KUKA KRL program: ps_602c3_bolha.src, ps_602c3_bolha.dat

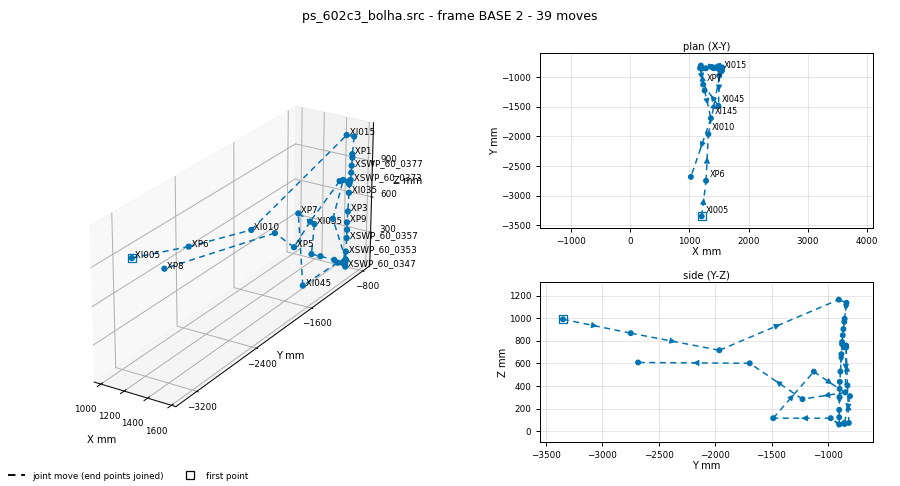
[picture p0: tool path of ps_602c3_bolha.src in frame BASE 2, 39 of 39 moves have a stored position in this frame; points joined in program order, loops and branches not executed]
--- ps_602c3_bolha.src ---
&ACCESS RVO1
&REL 1
&COMMENT Solda respot
&PARAM DISKPATH = KRC:\R1\Program
DEF ps_602c3_bolha( )

;FOLD INI
;FOLD SPOTTECH INI
USERSPOT(#INIT)
;ENDFOLD (SPOTTECH INI)
;FOLD GRIPPERTECH INI
USER_GRP(0,DUMMY,DUMMY,GDEFAULT)
;ENDFOLD (GRIPPERTECH INI)
  ;FOLD USER INI
    ;Make your modifications here

  ;ENDFOLD (USER INI)

   ;FOLD USER INI
      ;Make your modifications here
         ;FOLD COLLISION_V_3.01 INI
            IF (COLLISION_DATA[1].I_NR>0) THEN
               GLOBAL INTERRUPT DECL 21 WHEN $IN[COLLISION_DATA[1].I_NR]==FALSE DO COLLSTOP (1,0 )
            ENDIF
            IF (COLLISION_DATA[2].I_NR>0) THEN
               GLOBAL INTERRUPT DECL 22 WHEN $IN[COLLISION_DATA[2].I_NR]==FALSE DO COLLSTOP (2,0 )
            ENDIF
            IF (COLLISION_DATA[3].I_NR>0) THEN
               GLOBAL INTERRUPT DECL 23 WHEN $IN[COLLISION_DATA[3].I_NR]==FALSE DO COLLSTOP (3,0 )
            ENDIF
            IF (COLLISION_DATA[4].I_NR>0) THEN
               GLOBAL INTERRUPT DECL 24 WHEN $IN[COLLISION_DATA[4].I_NR]==FALSE DO COLLSTOP (4,0 )
            ENDIF
         ;ENDFOLD (COLLISION_V_3.01 INI)

   ;ENDFOLD (USER INI)
;ENDFOLD (INI)

; Caracterização dos meios de produção:
; Versão Atual:
; 15/05/2015 12:00 Name: P13.060-R1 CHANGES: Solda Geometrica Actros
; Gripper (INI;%{E}%V3.2.0,%MKUKATPGRIPPER,%CINIT,%VINIT,%P)

chk_w4_wechs_ok ( )           ; CHECK FERRAMENTA: C3

IF (NOT(GHOST())) THEN
IF MaxStandMenge (4) THEN
  MaxStandmengeErreicht (4)
ENDIF

IF Elektrodenwechsel (4) THEN
e_fraes_4()
ENDIF
ENDIF

;FOLD PTP l005  Vel=100 % P_OLP2 Tool[4]:Gun C03 Base[2]:Accelo;%{PE}%R8.2.20,%MKUKATPBASIS,%CMOVE,%VPTP,%P 1:PTP, 2:l005, 3:, 5:100, 7:P_OLP2
$BWDSTART = FALSE
PDAT_ACT= PP_OLP2
FDAT_ACT= Fl005
BAS(#PTP_PARAMS,100)
PTP Xl005
;ENDFOLD
;FOLD PTP P6 CONT Vel=100 % PDAT46 Tool[4]:PINCA C3 Base[2]:Accelo;%{PE}%R 8.2.20,%MKUKATPBASIS,%CMOVE,%VPTP,%P 1:PTP, 2:P6, 3:C_DIS, 5:100, 7:PDAT46
$BWDSTART=FALSE
PDAT_ACT=PPDAT46
FDAT_ACT=FP6
BAS(#PTP_PARAMS,100)
PTP XP6 C_DIS
;ENDFOLD
;FOLD PTP l010 Vel=100 % P_OLP3 Tool[4]:PINCA C3 Base[2]:Accelo;%{PE}%R 8.2.20,%MKUKATPBASIS,%CMOVE,%VPTP,%P 1:PTP, 2:l010, 3:, 5:100, 7:P_OLP3
$BWDSTART=FALSE
PDAT_ACT=PP_OLP3
FDAT_ACT=Fl010
BAS(#PTP_PARAMS,100)
PTP Xl010
;ENDFOLD

;FOLD OUT 3365 'R1_Solicita Lib. Soldar Geo1' State=TRUE ;%{PE}%R 8.2.20,%MKUKATPBASIS,%COUT,%VOUTX,%P 2:3365, 3:R1_Solicita Lib. Soldar Geo1, 5:TRUE, 6:
$OUT[3365]=TRUE
;ENDFOLD
;FOLD WAIT FOR ( IN 3323 'R1_Aguarda Lib. Soldar Respot GEO1' );%{PE}%R 8.2.20,%MKUKATPBASIS,%CEXT_WAIT_FOR,%VEXT_WAIT_FOR,%P 2:, 4:, 5:$IN, 6:3323, 7:R1_Aguarda Lib. Soldar Respot GEO1, 9:
WAIT FOR  ( $IN[3323] )
;ENDFOLD
;FOLD OUT 3331 'R1_Soldando' State=TRUE ;%{PE}%R 8.2.20,%MKUKATPBASIS,%COUT,%VOUTX,%P 2:3331, 3:R1_Soldando, 5:TRUE, 6:
$OUT[3331]=TRUE
;ENDFOLD
;FOLD OUT 3365 'R1_Solicita Lib. Soldar Geo1' State=FALSE ;%{PE}%R 8.2.20,%MKUKATPBASIS,%COUT,%VOUTX,%P 2:3365, 3:R1_Solicita Lib. Soldar Geo1, 5:FALSE, 6:
$OUT[3365]=FALSE
;ENDFOLD
;FOLD OUT 3369 'Area de Solda' State=FALSE ;%{PE}%R 8.2.20,%MKUKATPBASIS,%COUT,%VOUTX,%P 2:3369, 3:Area de Solda, 5:FALSE, 6:
$OUT[3369]=FALSE
;ENDFOLD

;FOLD PTP l015 CONT Vel=100 % PDAT1 Tool[4]:PINCA C3 Base[2]:Accelo;%{PE}%R 8.2.20,%MKUKATPBASIS,%CMOVE,%VPTP,%P 1:PTP, 2:l015, 3:C_DIS, 5:100, 7:PDAT1
$BWDSTART=FALSE
PDAT_ACT=PPDAT1
FDAT_ACT=Fl015
BAS(#PTP_PARAMS,100)
PTP Xl015 C_DIS
;ENDFOLD

;FOLD ; SWP_60_0385;%{PE}%R8.2.2,%MKUKATPSPOT,%CCOMMENT,%VNORMAL,%P 2:SWP_60_0385
;ENDFOLD
;FOLD PTP SWP_60_0385 PDAT2 SPOT Gun=3 RETR CLS PgNo1=151 ACTIVE=1 Tool[4]:PINCA C3 Base[2]:Accelo;%{PE}%R 8.2.2,%MKUKATPSPOT,%CSPOT,%VPTP,%P 1:PTP, 2:SWP_60_0385, 3:, 5:100, 7:PDAT2, 10:3, 12:#FIRST, 14:#CLO, 16:151, 18:1, 20:1, 22:0, 24:1, 25:NORMAL
$BWDSTART=FALSE
PDAT_ACT=PPDAT2
FDAT_ACT=FSWP_60_0385
BAS(#PTP_PARAMS,PPDAT2.VEL)
S_ACT.GUN=3
S_ACT.PAIR=SDEFAULT.PAIR
S_ACT.RETR=#CLO
S_ACT.CLO_TM=1
S_ACT.PGNO1=151
S_ACT.PGNO2=SDEFAULT.PGNO2
S_ACT.PRESS1=SDEFAULT.PRESS1
S_ACT.PRESS2=SDEFAULT.PRESS2
S_READY=FALSE
PTP XSWP_60_0385
USERSPOT(#SPOT, S_ACT)
WAIT FOR S_READY
;ENDFOLD

;FOLD PTP P1 CONT Vel=100 % PDAT7 Tool[4]:PINCA C3 Base[2]:Accelo;%{PE}%R 8.2.20,%MKUKATPBASIS,%CMOVE,%VPTP,%P 1:PTP, 2:P1, 3:C_DIS, 5:100, 7:PDAT7
$BWDSTART=FALSE
PDAT_ACT=PPDAT7
FDAT_ACT=FP1
BAS(#PTP_PARAMS,100)
PTP XP1 C_DIS
;ENDFOLD

;FOLD ; SWP_60_0379_1;%{PE}%R8.2.2,%MKUKATPSPOT,%CCOMMENT,%VNORMAL,%P 2:SWP_60_0379_1
;ENDFOLD
;FOLD PTP SWP_60_0379_1 PDAT6 SPOT Gun=3 RETR CLS PgNo1=153 ACTIVE=1 Tool[4]:PINCA C3 Base[2]:Accelo;%{PE}%R 8.2.2,%MKUKATPSPOT,%CSPOT,%VPTP,%P 1:PTP, 2:SWP_60_0379_1, 3:, 5:100, 7:PDAT6, 10:3, 12:#FIRST, 14:#CLO, 16:153, 18:1, 20:1, 22:0, 24:1, 25:NORMAL
$BWDSTART=FALSE
PDAT_ACT=PPDAT6
FDAT_ACT=FSWP_60_0379_1
BAS(#PTP_PARAMS,PPDAT6.VEL)
S_ACT.GUN=3
S_ACT.PAIR=SDEFAULT.PAIR
S_ACT.RETR=#CLO
S_ACT.CLO_TM=1
S_ACT.PGNO1=153
S_ACT.PGNO2=SDEFAULT.PGNO2
S_ACT.PRESS1=SDEFAULT.PRESS1
S_ACT.PRESS2=SDEFAULT.PRESS2
S_READY=FALSE
PTP XSWP_60_0379_1
USERSPOT(#SPOT, S_ACT)
WAIT FOR S_READY
;ENDFOLD

;FOLD ; SWP_60_0377;%{PE}%R8.2.2,%MKUKATPSPOT,%CCOMMENT,%VNORMAL,%P 2:SWP_60_0377
;ENDFOLD
;FOLD PTP SWP_60_0377 PDAT8 SPOT Gun=3 RETR CLS PgNo1=154 ACTIVE=1 Tool[4]:PINCA C3 Base[2]:Accelo;%{PE}%R 8.2.2,%MKUKATPSPOT,%CSPOT,%VPTP,%P 1:PTP, 2:SWP_60_0377, 3:, 5:100, 7:PDAT8, 10:3, 12:#FIRST, 14:#CLO, 16:154, 18:1, 20:1, 22:0, 24:1, 25:NORMAL
$BWDSTART=FALSE
PDAT_ACT=PPDAT8
FDAT_ACT=FSWP_60_0377
BAS(#PTP_PARAMS,PPDAT8.VEL)
S_ACT.GUN=3
S_ACT.PAIR=SDEFAULT.PAIR
S_ACT.RETR=#CLO
S_ACT.CLO_TM=1
S_ACT.PGNO1=154
S_ACT.PGNO2=SDEFAULT.PGNO2
S_ACT.PRESS1=SDEFAULT.PRESS1
S_ACT.PRESS2=SDEFAULT.PRESS2
S_READY=FALSE
PTP XSWP_60_0377
USERSPOT(#SPOT, S_ACT)
WAIT FOR S_READY
;ENDFOLD

;FOLD ; SWP_60_0375;%{PE}%R8.2.2,%MKUKATPSPOT,%CCOMMENT,%VNORMAL,%P 2:SWP_60_0375
;ENDFOLD
;FOLD PTP SWP_60_0375 PDAT9 SPOT Gun=3 RETR CLS PgNo1=155 ACTIVE=1 Tool[4]:PINCA C3 Base[2]:Accelo;%{PE}%R 8.2.2,%MKUKATPSPOT,%CSPOT,%VPTP,%P 1:PTP, 2:SWP_60_0375, 3:, 5:100, 7:PDAT9, 10:3, 12:#FIRST, 14:#CLO, 16:155, 18:1, 20:1, 22:0, 24:1, 25:NORMAL
$BWDSTART=FALSE
PDAT_ACT=PPDAT9
FDAT_ACT=FSWP_60_0375
BAS(#PTP_PARAMS,PPDAT9.VEL)
S_ACT.GUN=3
S_ACT.PAIR=SDEFAULT.PAIR
S_ACT.RETR=#CLO
S_ACT.CLO_TM=1
S_ACT.PGNO1=155
S_ACT.PGNO2=SDEFAULT.PGNO2
S_ACT.PRESS1=SDEFAULT.PRESS1
S_ACT.PRESS2=SDEFAULT.PRESS2
S_READY=FALSE
PTP XSWP_60_0375
USERSPOT(#SPOT, S_ACT)
WAIT FOR S_READY
;ENDFOLD

;FOLD ; SWP_60_0373;%{PE}%R8.2.2,%MKUKATPSPOT,%CCOMMENT,%VNORMAL,%P 2:SWP_60_0373
;ENDFOLD
;FOLD PTP SWP_60_0373 PDAT10 SPOT Gun=3 RETR CLS PgNo1=156 ACTIVE=1 Tool[4]:PINCA C3 Base[2]:Accelo;%{PE}%R 8.2.2,%MKUKATPSPOT,%CSPOT,%VPTP,%P 1:PTP, 2:SWP_60_0373, 3:, 5:100, 7:PDAT10, 10:3, 12:#FIRST, 14:#CLO, 16:156, 18:1, 20:1, 22:0, 24:1, 25:NORMAL
$BWDSTART=FALSE
PDAT_ACT=PPDAT10
FDAT_ACT=FSWP_60_0373
BAS(#PTP_PARAMS,PPDAT10.VEL)
S_ACT.GUN=3
S_ACT.PAIR=SDEFAULT.PAIR
S_ACT.RETR=#CLO
S_ACT.CLO_TM=1
S_ACT.PGNO1=156
S_ACT.PGNO2=SDEFAULT.PGNO2
S_ACT.PRESS1=SDEFAULT.PRESS1
S_ACT.PRESS2=SDEFAULT.PRESS2
S_READY=FALSE
PTP XSWP_60_0373
USERSPOT(#SPOT, S_ACT)
WAIT FOR S_READY
;ENDFOLD

;FOLD PTP P10 CONT Vel=100 % PDAT50 Tool[4]:PINCA C3 Base[2]:Accelo;%{PE}%R 8.2.20,%MKUKATPBASIS,%CMOVE,%VPTP,%P 1:PTP, 2:P10, 3:C_DIS, 5:100, 7:PDAT50
$BWDSTART=FALSE
PDAT_ACT=PPDAT50
FDAT_ACT=FP10
BAS(#PTP_PARAMS,100)
PTP XP10 C_DIS
;ENDFOLD
;FOLD PTP l035 CONT Vel=100 % PDAT11 Tool[4]:PINCA C3 Base[2]:Accelo;%{PE}%R 8.2.20,%MKUKATPBASIS,%CMOVE,%VPTP,%P 1:PTP, 2:l035, 3:C_DIS, 5:100, 7:PDAT11
$BWDSTART=FALSE
PDAT_ACT=PPDAT11
FDAT_ACT=Fl035
BAS(#PTP_PARAMS,100)
PTP Xl035 C_DIS
;ENDFOLD
;FOLD PTP P3 CONT Vel=100 % PDAT15 Tool[4]:PINCA C3 Base[2]:Accelo;%{PE}%R 8.2.20,%MKUKATPBASIS,%CMOVE,%VPTP,%P 1:PTP, 2:P3, 3:C_DIS, 5:100, 7:PDAT15
$BWDSTART=FALSE
PDAT_ACT=PPDAT15
FDAT_ACT=FP3
BAS(#PTP_PARAMS,100)
PTP XP3 C_DIS
;ENDFOLD
;FOLD PTP P9 CONT Vel=100 % PDAT49 Tool[4]:PINCA C3 Base[2]:Accelo;%{PE}%R 8.2.20,%MKUKATPBASIS,%CMOVE,%VPTP,%P 1:PTP, 2:P9, 3:C_DIS, 5:100, 7:PDAT49
$BWDSTART=FALSE
PDAT_ACT=PPDAT49
FDAT_ACT=FP9
BAS(#PTP_PARAMS,100)
PTP XP9 C_DIS
;ENDFOLD

;FOLD ; SWP_60_0359;%{PE}%R8.2.2,%MKUKATPSPOT,%CCOMMENT,%VNORMAL,%P 2:SWP_60_0359
;ENDFOLD
;FOLD PTP SWP_60_0359 PDAT16 SPOT Gun=3 RETR CLS PgNo1=158 ACTIVE=1 Tool[4]:PINCA C3 Base[2]:Accelo;%{PE}%R 8.2.2,%MKUKATPSPOT,%CSPOT,%VPTP,%P 1:PTP, 2:SWP_60_0359, 3:, 5:100, 7:PDAT16, 10:3, 12:#FIRST, 14:#CLO, 16:158, 18:1, 20:1, 22:0, 24:1, 25:NORMAL
$BWDSTART=FALSE
PDAT_ACT=PPDAT16
FDAT_ACT=FSWP_60_0359
BAS(#PTP_PARAMS,PPDAT16.VEL)
S_ACT.GUN=3
S_ACT.PAIR=SDEFAULT.PAIR
S_ACT.RETR=#CLO
S_ACT.CLO_TM=1
S_ACT.PGNO1=158
S_ACT.PGNO2=SDEFAULT.PGNO2
S_ACT.PRESS1=SDEFAULT.PRESS1
S_ACT.PRESS2=SDEFAULT.PRESS2
S_READY=FALSE
PTP XSWP_60_0359
USERSPOT(#SPOT, S_ACT)
WAIT FOR S_READY
;ENDFOLD

;FOLD ; SWP_60_0357;%{PE}%R8.2.2,%MKUKATPSPOT,%CCOMMENT,%VNORMAL,%P 2:SWP_60_0357
;ENDFOLD
;FOLD PTP SWP_60_0357 PDAT17 SPOT Gun=3 RETR CLS PgNo1=159 ACTIVE=1 Tool[4]:PINCA C3 Base[2]:Accelo;%{PE}%R 8.2.2,%MKUKATPSPOT,%CSPOT,%VPTP,%P 1:PTP, 2:SWP_60_0357, 3:, 5:100, 7:PDAT17, 10:3, 12:#FIRST, 14:#CLO, 16:159, 18:1, 20:1, 22:0, 24:1, 25:NORMAL
$BWDSTART=FALSE
PDAT_ACT=PPDAT17
FDAT_ACT=FSWP_60_0357
BAS(#PTP_PARAMS,PPDAT17.VEL)
S_ACT.GUN=3
S_ACT.PAIR=SDEFAULT.PAIR
S_ACT.RETR=#CLO
S_ACT.CLO_TM=1
S_ACT.PGNO1=159
S_ACT.PGNO2=SDEFAULT.PGNO2
S_ACT.PRESS1=SDEFAULT.PRESS1
S_ACT.PRESS2=SDEFAULT.PRESS2
S_READY=FALSE
PTP XSWP_60_0357
USERSPOT(#SPOT, S_ACT)
WAIT FOR S_READY
;ENDFOLD

;FOLD ; SWP_60_0353;%{PE}%R8.2.2,%MKUKATPSPOT,%CCOMMENT,%VNORMAL,%P 2:SWP_60_0353
;ENDFOLD
;FOLD PTP SWP_60_0353 PDAT18 SPOT Gun=3 RETR CLS PgNo1=160 ACTIVE=1 Tool[4]:PINCA C3 Base[2]:Accelo;%{PE}%R 8.2.2,%MKUKATPSPOT,%CSPOT,%VPTP,%P 1:PTP, 2:SWP_60_0353, 3:, 5:100, 7:PDAT18, 10:3, 12:#FIRST, 14:#CLO, 16:160, 18:1, 20:1, 22:0, 24:1, 25:NORMAL
$BWDSTART=FALSE
PDAT_ACT=PPDAT18
FDAT_ACT=FSWP_60_0353
BAS(#PTP_PARAMS,PPDAT18.VEL)
S_ACT.GUN=3
S_ACT.PAIR=SDEFAULT.PAIR
S_ACT.RETR=#CLO
S_ACT.CLO_TM=1
S_ACT.PGNO1=160
S_ACT.PGNO2=SDEFAULT.PGNO2
S_ACT.PRESS1=SDEFAULT.PRESS1
S_ACT.PRESS2=SDEFAULT.PRESS2
S_READY=FALSE
PTP XSWP_60_0353
USERSPOT(#SPOT, S_ACT)
WAIT FOR S_READY
;ENDFOLD

;FOLD ; SWP_60_0351;%{PE}%R8.2.2,%MKUKATPSPOT,%CCOMMENT,%VNORMAL,%P 2:SWP_60_0351
;ENDFOLD
;FOLD PTP SWP_60_0351 PDAT19 SPOT Gun=3 RETR CLS PgNo1=161 ACTIVE=1 Tool[4]:PINCA C3 Base[2]:Accelo;%{PE}%R 8.2.2,%MKUKATPSPOT,%CSPOT,%VPTP,%P 1:PTP, 2:SWP_60_0351, 3:, 5:100, 7:PDAT19, 10:3, 12:#FIRST, 14:#CLO, 16:161, 18:1, 20:1, 22:0, 24:1, 25:NORMAL
$BWDSTART=FALSE
PDAT_ACT=PPDAT19
FDAT_ACT=FSWP_60_0351
BAS(#PTP_PARAMS,PPDAT19.VEL)
S_ACT.GUN=3
S_ACT.PAIR=SDEFAULT.PAIR
S_ACT.RETR=#CLO
S_ACT.CLO_TM=1
S_ACT.PGNO1=161
S_ACT.PGNO2=SDEFAULT.PGNO2
S_ACT.PRESS1=SDEFAULT.PRESS1
S_ACT.PRESS2=SDEFAULT.PRESS2
S_READY=FALSE
PTP XSWP_60_0351
USERSPOT(#SPOT, S_ACT)
WAIT FOR S_READY
;ENDFOLD

;FOLD ; SWP_60_0347;%{PE}%R8.2.2,%MKUKATPSPOT,%CCOMMENT,%VNORMAL,%P 2:SWP_60_0347
;ENDFOLD
;FOLD PTP SWP_60_0347 PDAT20 SPOT Gun=3 RETR OPN PgNo1=162 ACTIVE=1 Tool[4]:PINCA C3 Base[2]:Accelo;%{PE}%R 8.2.2,%MKUKATPSPOT,%CSPOT,%VPTP,%P 1:PTP, 2:SWP_60_0347, 3:, 5:100, 7:PDAT20, 10:3, 12:#FIRST, 14:#OPN, 16:162, 18:1, 20:0, 22:0, 24:1, 25:NORMAL
$BWDSTART=FALSE
PDAT_ACT=PPDAT20
FDAT_ACT=FSWP_60_0347
BAS(#PTP_PARAMS,PPDAT20.VEL)
S_ACT.GUN=3
S_ACT.PAIR=SDEFAULT.PAIR
S_ACT.RETR=#OPN
S_ACT.CLO_TM=1
S_ACT.PGNO1=162
S_ACT.PGNO2=SDEFAULT.PGNO2
S_ACT.PRESS1=SDEFAULT.PRESS1
S_ACT.PRESS2=SDEFAULT.PRESS2
S_READY=FALSE
PTP XSWP_60_0347
USERSPOT(#SPOT, S_ACT)
WAIT FOR S_READY
;ENDFOLD

;FOLD PTP l040 CONT Vel=100 % PDAT21 Tool[4]:PINCA C3 Base[2]:Accelo;%{PE}%R 8.2.20,%MKUKATPBASIS,%CMOVE,%VPTP,%P 1:PTP, 2:l040, 3:C_DIS, 5:100, 7:PDAT21
$BWDSTART=FALSE
PDAT_ACT=PPDAT21
FDAT_ACT=Fl040
BAS(#PTP_PARAMS,100)
PTP Xl040 C_DIS
;ENDFOLD
;FOLD PTP l045 Vel=100 % PDAT22 Tool[4]:PINCA C3 Base[2]:Accelo;%{PE}%R 8.2.20,%MKUKATPBASIS,%CMOVE,%VPTP,%P 1:PTP, 2:l045, 3:, 5:100, 7:PDAT22
$BWDSTART=FALSE
PDAT_ACT=PPDAT22
FDAT_ACT=Fl045
BAS(#PTP_PARAMS,100)
PTP Xl045
;ENDFOLD

;FOLD Collision.Monitoring_3_On ;%{PE}%MKUKATPUSER
COLLSTOP( 3, 1 ) ;Interrupt-Controlled
;ENDFOLD

;FOLD PTP P7 CONT Vel=100 % PDAT47 Tool[4]:PINCA C3 Base[2]:Accelo;%{PE}%R 8.2.20,%MKUKATPBASIS,%CMOVE,%VPTP,%P 1:PTP, 2:P7, 3:C_DIS, 5:100, 7:PDAT47
$BWDSTART=FALSE
PDAT_ACT=PPDAT47
FDAT_ACT=FP7
BAS(#PTP_PARAMS,100)
PTP XP7 C_DIS
;ENDFOLD
;FOLD PTP l055 CONT Vel=100 % PDAT23 Tool[4]:PINCA C3 Base[2]:Accelo;%{PE}%R 8.2.20,%MKUKATPBASIS,%CMOVE,%VPTP,%P 1:PTP, 2:l055, 3:C_DIS, 5:100, 7:PDAT23
$BWDSTART=FALSE
PDAT_ACT=PPDAT23
FDAT_ACT=Fl055
BAS(#PTP_PARAMS,100)
PTP Xl055 C_DIS
;ENDFOLD

;FOLD ; SWP_60_0329;%{PE}%R8.2.2,%MKUKATPSPOT,%CCOMMENT,%VNORMAL,%P 2:SWP_60_0329
;ENDFOLD
;FOLD PTP SWP_60_0329 PDAT25 SPOT Gun=3 RETR CLS PgNo1=163 ACTIVE=1 Tool[4]:PINCA C3 Base[2]:Accelo;%{PE}%R 8.2.2,%MKUKATPSPOT,%CSPOT,%VPTP,%P 1:PTP, 2:SWP_60_0329, 3:, 5:100, 7:PDAT25, 10:3, 12:#FIRST, 14:#CLO, 16:163, 18:1, 20:0, 22:0, 24:1, 25:NORMAL
$BWDSTART=FALSE
PDAT_ACT=PPDAT25
FDAT_ACT=FSWP_60_0329
BAS(#PTP_PARAMS,PPDAT25.VEL)
S_ACT.GUN=3
S_ACT.PAIR=SDEFAULT.PAIR
S_ACT.RETR=#CLO
S_ACT.CLO_TM=1
S_ACT.PGNO1=163
S_ACT.PGNO2=SDEFAULT.PGNO2
S_ACT.PRESS1=SDEFAULT.PRESS1
S_ACT.PRESS2=SDEFAULT.PRESS2
S_READY=FALSE
PTP XSWP_60_0329
USERSPOT(#SPOT, S_ACT)
WAIT FOR S_READY
;ENDFOLD

;FOLD PTP l065 CONT Vel=100 % PDAT26 Tool[4]:PINCA C3 Base[2]:Accelo;%{PE}%R 8.2.20,%MKUKATPBASIS,%CMOVE,%VPTP,%P 1:PTP, 2:l065, 3:C_DIS, 5:100, 7:PDAT26
$BWDSTART=FALSE
PDAT_ACT=PPDAT26
FDAT_ACT=Fl065
BAS(#PTP_PARAMS,100)
PTP Xl065 C_DIS
;ENDFOLD
;FOLD PTP l070 CONT Vel=100 % PDAT27 Tool[4]:PINCA C3 Base[2]:Accelo;%{PE}%R 8.2.20,%MKUKATPBASIS,%CMOVE,%VPTP,%P 1:PTP, 2:l070, 3:C_DIS, 5:100, 7:PDAT27
$BWDSTART=FALSE
PDAT_ACT=PPDAT27
FDAT_ACT=Fl070
BAS(#PTP_PARAMS,100)
PTP Xl070 C_DIS
;ENDFOLD

;FOLD ; SWP_60_0343;%{PE}%R8.2.2,%MKUKATPSPOT,%CCOMMENT,%VNORMAL,%P 2:SWP_60_0343
;ENDFOLD
;FOLD PTP SWP_60_0343 PDAT28 SPOT Gun=3 RETR CLS PgNo1=165 ACTIVE=1 Tool[4]:PINCA C3 Base[2]:Accelo;%{PE}%R 8.2.2,%MKUKATPSPOT,%CSPOT,%VPTP,%P 1:PTP, 2:SWP_60_0343, 3:, 5:100, 7:PDAT28, 10:3, 12:#FIRST, 14:#CLO, 16:165, 18:1, 20:0, 22:0, 24:1, 25:NORMAL
$BWDSTART=FALSE
PDAT_ACT=PPDAT28
FDAT_ACT=FSWP_60_0343
BAS(#PTP_PARAMS,PPDAT28.VEL)
S_ACT.GUN=3
S_ACT.PAIR=SDEFAULT.PAIR
S_ACT.RETR=#CLO
S_ACT.CLO_TM=1
S_ACT.PGNO1=165
S_ACT.PGNO2=SDEFAULT.PGNO2
S_ACT.PRESS1=SDEFAULT.PRESS1
S_ACT.PRESS2=SDEFAULT.PRESS2
S_READY=FALSE
PTP XSWP_60_0343
USERSPOT(#SPOT, S_ACT)
WAIT FOR S_READY
;ENDFOLD

;FOLD ; SWP_60_0345;%{PE}%R8.2.2,%MKUKATPSPOT,%CCOMMENT,%VNORMAL,%P 2:SWP_60_0345
;ENDFOLD
;FOLD PTP SWP_60_0345 PDAT29 SPOT Gun=3 RETR OPN PgNo1=164 ACTIVE=1 Tool[4]:PINCA C3 Base[2]:Accelo;%{PE}%R 8.2.2,%MKUKATPSPOT,%CSPOT,%VPTP,%P 1:PTP, 2:SWP_60_0345, 3:, 5:100, 7:PDAT29, 10:3, 12:#FIRST, 14:#OPN, 16:164, 18:1, 20:0, 22:0, 24:1, 25:NORMAL
$BWDSTART=FALSE
PDAT_ACT=PPDAT29
FDAT_ACT=FSWP_60_0345
BAS(#PTP_PARAMS,PPDAT29.VEL)
S_ACT.GUN=3
S_ACT.PAIR=SDEFAULT.PAIR
S_ACT.RETR=#OPN
S_ACT.CLO_TM=1
S_ACT.PGNO1=164
S_ACT.PGNO2=SDEFAULT.PGNO2
S_ACT.PRESS1=SDEFAULT.PRESS1
S_ACT.PRESS2=SDEFAULT.PRESS2
S_READY=FALSE
PTP XSWP_60_0345
USERSPOT(#SPOT, S_ACT)
WAIT FOR S_READY
;ENDFOLD

;FOLD PTP l075 CONT Vel=100 % PDAT30 Tool[4]:PINCA C3 Base[2]:Accelo;%{PE}%R 8.2.20,%MKUKATPBASIS,%CMOVE,%VPTP,%P 1:PTP, 2:l075, 3:C_DIS, 5:100, 7:PDAT30
$BWDSTART=FALSE
PDAT_ACT=PPDAT30
FDAT_ACT=Fl075
BAS(#PTP_PARAMS,100)
PTP Xl075 C_DIS
;ENDFOLD
;FOLD PTP l080 CONT Vel=100 % PDAT31 Tool[4]:PINCA C3 Base[2]:Accelo;%{PE}%R 8.2.20,%MKUKATPBASIS,%CMOVE,%VPTP,%P 1:PTP, 2:l080, 3:C_DIS, 5:100, 7:PDAT31
$BWDSTART=FALSE
PDAT_ACT=PPDAT31
FDAT_ACT=Fl080
BAS(#PTP_PARAMS,100)
PTP Xl080 C_DIS
;ENDFOLD
;FOLD PTP l110 CONT Vel=100 % PDAT39 Tool[4]:PINCA C3 Base[2]:Accelo;%{PE}%R 8.2.20,%MKUKATPBASIS,%CMOVE,%VPTP,%P 1:PTP, 2:l110, 3:C_DIS, 5:100, 7:PDAT39
$BWDSTART=FALSE
PDAT_ACT=PPDAT39
FDAT_ACT=Fl110
BAS(#PTP_PARAMS,100)
PTP Xl110 C_DIS
;ENDFOLD
;FOLD PTP l115 CONT Vel=100 % PDAT40 Tool[4]:PINCA C3 Base[2]:Accelo;%{PE}%R 8.2.20,%MKUKATPBASIS,%CMOVE,%VPTP,%P 1:PTP, 2:l115, 3:C_DIS, 5:100, 7:PDAT40
$BWDSTART=FALSE
PDAT_ACT=PPDAT40
FDAT_ACT=Fl115
BAS(#PTP_PARAMS,100)
PTP Xl115 C_DIS
;ENDFOLD

;FOLD ; SWP_60_0401;%{PE}%R8.2.2,%MKUKATPSPOT,%CCOMMENT,%VNORMAL,%P 2:SWP_60_0401
;ENDFOLD
;FOLD PTP SWP_60_0401 PDAT41 SPOT Gun=3 RETR OPN PgNo1=168 ACTIVE=1 Tool[4]:PINCA C3 Base[2]:Accelo;%{PE}%R 8.2.2,%MKUKATPSPOT,%CSPOT,%VPTP,%P 1:PTP, 2:SWP_60_0401, 3:, 5:100, 7:PDAT41, 10:3, 12:#FIRST, 14:#OPN, 16:168, 18:1, 20:0, 22:0, 24:1, 25:NORMAL
$BWDSTART=FALSE
PDAT_ACT=PPDAT41
FDAT_ACT=FSWP_60_0401
BAS(#PTP_PARAMS,PPDAT41.VEL)
S_ACT.GUN=3
S_ACT.PAIR=SDEFAULT.PAIR
S_ACT.RETR=#OPN
S_ACT.CLO_TM=1
S_ACT.PGNO1=168
S_ACT.PGNO2=SDEFAULT.PGNO2
S_ACT.PRESS1=SDEFAULT.PRESS1
S_ACT.PRESS2=SDEFAULT.PRESS2
S_READY=FALSE
PTP XSWP_60_0401
USERSPOT(#SPOT, S_ACT)
WAIT FOR S_READY
;ENDFOLD

;FOLD PTP l120 CONT Vel=100 % PDAT42 Tool[4]:PINCA C3 Base[2]:Accelo;%{PE}%R 8.2.20,%MKUKATPBASIS,%CMOVE,%VPTP,%P 1:PTP, 2:l120, 3:C_DIS, 5:100, 7:PDAT42
$BWDSTART=FALSE
PDAT_ACT=PPDAT42
FDAT_ACT=Fl120
BAS(#PTP_PARAMS,100)
PTP Xl120 C_DIS
;ENDFOLD
;FOLD PTP l125 CONT Vel=100 % PDAT43 Tool[4]:PINCA C3 Base[2]:Accelo;%{PE}%R 8.2.20,%MKUKATPBASIS,%CMOVE,%VPTP,%P 1:PTP, 2:l125, 3:C_DIS, 5:100, 7:PDAT43
$BWDSTART=FALSE
PDAT_ACT=PPDAT43
FDAT_ACT=Fl125
BAS(#PTP_PARAMS,100)
PTP Xl125 C_DIS
;ENDFOLD
;FOLD PTP l135 CONT Vel=100 % P_OLP6 Tool[4]:PINCA C3 Base[2]:Accelo;%{PE}%R 8.2.20,%MKUKATPBASIS,%CMOVE,%VPTP,%P 1:PTP, 2:l135, 3:C_DIS, 5:100, 7:P_OLP6
$BWDSTART=FALSE
PDAT_ACT=PP_OLP6
FDAT_ACT=Fl135
BAS(#PTP_PARAMS,100)
PTP Xl135 C_DIS
;ENDFOLD
;FOLD PTP P5 CONT Vel=100 % PDAT45 Tool[4]:PINCA C3 Base[2]:Accelo;%{PE}%R 8.2.20,%MKUKATPBASIS,%CMOVE,%VPTP,%P 1:PTP, 2:P5, 3:C_DIS, 5:100, 7:PDAT45
$BWDSTART=FALSE
PDAT_ACT=PPDAT45
FDAT_ACT=FP5
BAS(#PTP_PARAMS,100)
PTP XP5 C_DIS
;ENDFOLD
;FOLD PTP l145 CONT Vel=100 % P_OLP8 Tool[4]:PINCA C3 Base[2]:Accelo;%{PE}%R 8.2.20,%MKUKATPBASIS,%CMOVE,%VPTP,%P 1:PTP, 2:l145, 3:C_DIS, 5:100, 7:P_OLP8
$BWDSTART=FALSE
PDAT_ACT=PP_OLP8
FDAT_ACT=Fl145
BAS(#PTP_PARAMS,100)
PTP Xl145 C_DIS
;ENDFOLD

;FOLD OUT 3331 'R1_Soldando' State=FALSE ;%{PE}%R 8.2.20,%MKUKATPBASIS,%COUT,%VOUTX,%P 2:3331, 3:R1_Soldando, 5:FALSE, 6:
$OUT[3331]=FALSE
;ENDFOLD
;FOLD OUT 3369 'Area de Solda' State=TRUE ;%{PE}%R 8.2.20,%MKUKATPBASIS,%COUT,%VOUTX,%P 2:3369, 3:Area de Solda, 5:TRUE, 6:
$OUT[3369]=TRUE
;ENDFOLD

;FOLD PULSE 3367 'R1_Solda Respot Geo1 OK' State=TRUE Time=3 sec;%{PE}%R 8.2.20,%MKUKATPBASIS,%COUT,%VPULSE,%P 2:3367, 3:R1_Solda Respot Geo1 OK, 5:TRUE, 6:, 8:3
PULSE($OUT[3367], TRUE,3)
;ENDFOLD

;FOLD PTP P8 Vel=100 % PDAT48 Tool[4]:PINCA C3 Base[2]:Accelo;%{PE}%R 8.2.20,%MKUKATPBASIS,%CMOVE,%VPTP,%P 1:PTP, 2:P8, 3:, 5:100, 7:PDAT48
$BWDSTART=FALSE
PDAT_ACT=PPDAT48
FDAT_ACT=FP8
BAS(#PTP_PARAMS,100)
PTP XP8
;ENDFOLD

IF (NOT(GHOST())) THEN
IF FraesAnf(4) THEN
f_fraes_4()
ENDIF
ENDIF

END

--- ps_602c3_bolha.dat ---
&ACCESS RVO1
&REL 1
&COMMENT Solda respot
&PARAM DISKPATH = KRC:\R1\Program
DEFDAT  ps_602c3_bolha
;FOLD EXTERNAL DECLARATIONS;%{PE}%MKUKATPBASIS,%CEXT,%VCOMMON,%P
;FOLD GRIPPERTECH EXT
EXT  H50 (INT  :IN,INT  :IN,INT  :IN,GRP_TYP  :IN )
;ENDFOLD (GRIPPERTECH EXT)
;FOLD SPOTTECH EXT
EXT  USERSPOT (S_COMMAND  :IN,SPOT_TYPE  :IN )
;ENDFOLD (SPOTTECH EXT)
;FOLD BASISTECH EXT;%{PE}%MKUKATPBASIS,%CEXT,%VEXT,%P
EXT  BAS (BAS_COMMAND  :IN,REAL  :IN )
DECL INT SUCCESS
;ENDFOLD (BASISTECH EXT)
;FOLD USER EXT;%{E}%MKUKATPUSER,%CEXT,%VEXT,%P
;Make your modifications here

;ENDFOLD (USER EXT)
;ENDFOLD (EXTERNAL DECLARATIONS)
DECL FDAT FLO1077={TOOL_NO 4,BASE_NO 2,IPO_FRAME #BASE,POINT2[] " "}
DECL PDAT PP_OLP1={VEL 100.0,ACC 50.0,APO_DIST 0.0}
DECL FDAT Fl005={TOOL_NO 4,BASE_NO 2,IPO_FRAME #BASE,POINT2[] " "}
DECL PDAT PP_OLP2={VEL 100.0,ACC 50.0,APO_DIST 0.0}
DECL E6POS Xl005={X 1207.93994,Y -3347.26807,Z 991.342712,A 123.692596,B -61.2644691,C 128.996994,S 18,T 3,E1 0.0,E2 0.0,E3 0.0,E4 0.0,E5 0.0,E6 0.0}
DECL FDAT Fl010={TOOL_NO 4,BASE_NO 2,IPO_FRAME #BASE,POINT2[] " "}
DECL PDAT PP_OLP3={VEL 100.0,ACC 100.0,APO_DIST 10.0,APO_MODE #CDIS}
DECL E6POS Xl010={X 1321.125,Y -1961.92896,Z 716.955383,A 162.414505,B -50.7519913,C 56.327549,S 18,T 3,E1 0.0,E2 0.0,E3 0.0,E4 0.0,E5 0.0,E6 0.0}
DECL FDAT Fl015={TOOL_NO 4,BASE_NO 2,IPO_FRAME #BASE,POINT2[] " "}
DECL E6POS Xl015={X 1525.30005,Y -903.920776,Z 1165.68701,A 79.9386902,B -67.3189468,C 102.332298,S 18,T 3,E1 0.0,E2 0.0,E3 0.0,E4 0.0,E5 0.0,E6 0.0}
DECL LDAT LL_OLP1={VEL 2.0,ACC 23.0,APO_DIST 0.0,APO_FAC 0.0,ORI_TYP #VAR,CIRC_TYP #BASE,JERK_FAC 50.0}
DECL FDAT FSWP_60_0387={TOOL_NO 4,BASE_NO 2,IPO_FRAME #BASE,POINT2[] " ",TQ_STATE FALSE}
DECL E6POS XSWP_60_0387={X 1552.93799,Y -826.98468,Z 1187.58105,A 86.6566467,B -69.5555801,C 96.031723,S 18,T 3,E1 0.0,E2 0.0,E3 0.0,E4 0.0,E5 0.0,E6 0.0}
DECL LDAT LL_OLP2={VEL 2.0,ACC 23.0,APO_DIST 0.0,APO_FAC 0.0,ORI_TYP #VAR,CIRC_TYP #BASE,JERK_FAC 50.0}
DECL FDAT FSWP_60_0385={TOOL_NO 4,BASE_NO 2,IPO_FRAME #BASE,POINT2[] " "}
DECL E6POS XSWP_60_0385={X 1553.06104,Y -835.943176,Z 1137.59094,A 86.8311081,B -70.8715897,C 95.7938004,S 18,T 3,E1 0.0,E2 0.0,E3 0.0,E4 0.0,E5 0.0,E6 0.0}
DECL LDAT LL_OLP3={VEL 2.0,ACC 23.0,APO_DIST 0.0,APO_FAC 0.0,ORI_TYP #VAR,CIRC_TYP #BASE,JERK_FAC 50.0}
DECL FDAT Fl020={TOOL_NO 4,BASE_NO 2,IPO_FRAME #BASE,POINT2[] " "}
DECL E6POS Xl020={X 1551.22803,Y -845.641479,Z 1079.81299,A 86.8358231,B -70.8698883,C 95.7901917,S 18,T 3,E1 0.0,E2 0.0,E3 0.0,E4 0.0,E5 0.0,E6 0.0}
DECL LDAT LL_OLP4={VEL 2.0,ACC 23.0,APO_DIST 0.0,APO_FAC 0.0,ORI_TYP #VAR,CIRC_TYP #BASE,JERK_FAC 50.0}
DECL FDAT Fl025={TOOL_NO 4,BASE_NO 2,IPO_FRAME #BASE,POINT2[] " "}
DECL E6POS Xl025={X 1489.18604,Y -870.828003,Z 1017.263,A -85.5016022,B 64.9662018,C -88.5036011,S 2,T 3}
DECL LDAT LL_OLP5={VEL 2.0,ACC 23.0,APO_DIST 0.0,APO_FAC 0.0,ORI_TYP #VAR,CIRC_TYP #BASE,JERK_FAC 50.0}
DECL FDAT FSWP_60_0381={TOOL_NO 4,BASE_NO 2,IPO_FRAME #BASE,POINT2[] " "}
DECL E6POS XSWP_60_0381={X 1553.82996,Y -848.580627,Z 1024.89001,A 86.8347931,B -70.8682632,C 95.7921371,S 18,T 3,E1 0.0,E2 0.0,E3 0.0,E4 0.0,E5 0.0,E6 0.0}
DECL LDAT LL_OLP6={VEL 2.0,ACC 23.0,APO_DIST 0.0,APO_FAC 0.0,ORI_TYP #VAR,CIRC_TYP #BASE,JERK_FAC 50.0}
DECL FDAT FSWP_60_0379_1={TOOL_NO 4,BASE_NO 2,IPO_FRAME #BASE,POINT2[] " "}
DECL E6POS XSWP_60_0379_1={X 1552.61804,Y -854.997192,Z 968.952271,A 94.1828384,B -64.9687424,C 88.8215866,S 18,T 3,E1 0.0,E2 0.0,E3 0.0,E4 0.0,E5 0.0,E6 0.0}
DECL LDAT LL_OLP7={VEL 2.0,ACC 23.0,APO_DIST 0.0,APO_FAC 0.0,ORI_TYP #VAR,CIRC_TYP #BASE,JERK_FAC 50.0}
DECL FDAT FSWP_60_0377={TOOL_NO 4,BASE_NO 2,IPO_FRAME #BASE,POINT2[] " "}
DECL E6POS XSWP_60_0377={X 1552.30103,Y -863.091309,Z 904.84729,A 93.829483,B -64.9712296,C 89.1674271,S 18,T 3,E1 0.0,E2 0.0,E3 0.0,E4 0.0,E5 0.0,E6 0.0}
DECL LDAT LL_OLP8={VEL 2.0,ACC 23.0,APO_DIST 0.0,APO_FAC 0.0,ORI_TYP #VAR,CIRC_TYP #BASE,JERK_FAC 50.0}
DECL FDAT FSWP_60_0375={TOOL_NO 4,BASE_NO 2,IPO_FRAME #BASE,POINT2[] " ",TQ_STATE FALSE}
DECL E6POS XSWP_60_0375={X 1552.65796,Y -868.826172,Z 849.536316,A 93.6191864,B -64.9780884,C 89.4089432,S 18,T 3,E1 0.0,E2 0.0,E3 0.0,E4 0.0,E5 0.0,E6 0.0}
DECL LDAT LL_OLP9={VEL 2.0,ACC 23.0,APO_DIST 0.0,APO_FAC 0.0,ORI_TYP #VAR,CIRC_TYP #BASE,JERK_FAC 50.0}
DECL FDAT FSWP_60_0373={TOOL_NO 4,BASE_NO 2,IPO_FRAME #BASE,POINT2[] " "}
DECL E6POS XSWP_60_0373={X 1551.63501,Y -874.4599,Z 790.400818,A 93.4071732,B -64.9728928,C 89.6387329,S 18,T 3,E1 0.0,E2 0.0,E3 0.0,E4 0.0,E5 0.0,E6 0.0}
DECL LDAT LL_OLP10={VEL 2.0,ACC 23.0,APO_DIST 0.0,APO_FAC 0.0,ORI_TYP #VAR,CIRC_TYP #BASE,JERK_FAC 50.0}
DECL FDAT Fl030={TOOL_NO 4,BASE_NO 2,IPO_FRAME #BASE,POINT2[] " "}
DECL E6POS Xl030={X 1492.099,Y -895.401978,Z 779.09198,A 93.4092026,B -64.9731979,C 89.6371002,S 2,T 3}
DECL LDAT LL_OLP11={VEL 2.0,ACC 23.0,APO_DIST 0.0,APO_FAC 0.0,ORI_TYP #VAR,CIRC_TYP #BASE,JERK_FAC 50.0}
DECL FDAT Fl035={TOOL_NO 4,BASE_NO 2,IPO_FRAME #BASE,POINT2[] " ",TQ_STATE FALSE}
DECL E6POS Xl035={X 1542.96594,Y -880.71698,Z 682.375793,A 93.1003113,B -57.6212807,C 89.9753418,S 18,T 3,E1 0.0,E2 0.0,E3 0.0,E4 0.0,E5 0.0,E6 0.0}
DECL LDAT LL_OLP12={VEL 2.0,ACC 23.0,APO_DIST 0.0,APO_FAC 0.0,ORI_TYP #VAR,CIRC_TYP #BASE,JERK_FAC 50.0}
DECL FDAT FSWP_60_0361={TOOL_NO 4,BASE_NO 2,IPO_FRAME #BASE,POINT2[] " "}
DECL E6POS XSWP_60_0361={X 1544.04797,Y -894.937378,Z 437.406708,A 92.7001419,B -40.9681511,C 90.4352493,S 18,T 3,E1 0.0,E2 0.0,E3 0.0,E4 0.0,E5 0.0,E6 0.0}
DECL LDAT LL_OLP13={VEL 2.0,ACC 23.0,APO_DIST 0.0,APO_FAC 0.0,ORI_TYP #VAR,CIRC_TYP #BASE,JERK_FAC 50.0}
DECL FDAT FSWP_60_0359={TOOL_NO 4,BASE_NO 2,IPO_FRAME #BASE,POINT2[] " "}
DECL E6POS XSWP_60_0359={X 1542.51099,Y -896.768372,Z 375.472687,A 92.7003326,B -40.9718399,C 90.4242401,S 18,T 3,E1 0.0,E2 0.0,E3 0.0,E4 0.0,E5 0.0,E6 0.0}
DECL LDAT LL_OLP14={VEL 2.0,ACC 23.0,APO_DIST 0.0,APO_FAC 0.0,ORI_TYP #VAR,CIRC_TYP #BASE,JERK_FAC 50.0}
DECL FDAT FSWP_60_0357={TOOL_NO 4,BASE_NO 2,IPO_FRAME #BASE,POINT2[] " "}
DECL E6POS XSWP_60_0357={X 1540.20203,Y -897.218506,Z 304.370087,A 92.751709,B -40.9723511,C 90.3579712,S 18,T 3,E1 0.0,E2 0.0,E3 0.0,E4 0.0,E5 0.0,E6 0.0}
DECL LDAT LL_OLP15={VEL 2.0,ACC 23.0,APO_DIST 0.0,APO_FAC 0.0,ORI_TYP #VAR,CIRC_TYP #BASE,JERK_FAC 50.0}
DECL FDAT FSWP_60_0353={TOOL_NO 4,BASE_NO 2,IPO_FRAME #BASE,POINT2[] " "}
DECL E6POS XSWP_60_0353={X 1537.75598,Y -900.391785,Z 189.053696,A 92.9539566,B -40.9735718,C 90.0922623,S 18,T 3,E1 0.0,E2 0.0,E3 0.0,E4 0.0,E5 0.0,E6 0.0}
DECL LDAT LL_OLP16={VEL 2.0,ACC 23.0,APO_DIST 0.0,APO_FAC 0.0,ORI_TYP #VAR,CIRC_TYP #BASE,JERK_FAC 50.0}
DECL FDAT FSWP_60_0351={TOOL_NO 4,BASE_NO 2,IPO_FRAME #BASE,POINT2[] " "}
DECL E6POS XSWP_60_0351={X 1535.66101,Y -900.398376,Z 123.525497,A 92.9552002,B -40.9745598,C 90.0935669,S 18,T 3,E1 0.0,E2 0.0,E3 0.0,E4 0.0,E5 0.0,E6 0.0}
DECL LDAT LL_OLP17={VEL 2.0,ACC 23.0,APO_DIST 0.0,APO_FAC 0.0,ORI_TYP #VAR,CIRC_TYP #BASE,JERK_FAC 50.0}
DECL FDAT FSWP_60_0347={TOOL_NO 4,BASE_NO 2,IPO_FRAME #BASE,POINT2[] " "}
DECL E6POS XSWP_60_0347={X 1534.60498,Y -899.584778,Z 59.1992111,A 93.1186523,B -40.9753189,C 89.8627701,S 18,T 3,E1 0.0,E2 0.0,E3 0.0,E4 0.0,E5 0.0,E6 0.0}
DECL LDAT LL_OLP18={VEL 2.0,ACC 23.0,APO_DIST 0.0,APO_FAC 0.0,ORI_TYP #VAR,CIRC_TYP #BASE,JERK_FAC 50.0}
DECL FDAT Fl040={TOOL_NO 4,BASE_NO 2,IPO_FRAME #BASE,POINT2[] " "}
DECL E6POS Xl040={X 1505.98804,Y -975.236206,Z 115.411598,A 93.1220627,B -40.9728699,C 89.8605804,S 18,T 3,E1 0.0,E2 0.0,E3 0.0,E4 0.0,E5 0.0,E6 0.0}
DECL LDAT LL_OLP19={VEL 2.0,ACC 23.0,APO_DIST 0.0,APO_FAC 0.0,ORI_TYP #VAR,CIRC_TYP #BASE,JERK_FAC 50.0}
DECL FDAT Fl045={TOOL_NO 4,BASE_NO 2,IPO_FRAME #BASE,POINT2[] " "}
DECL E6POS Xl045={X 1491.74402,Y -1485.05505,Z 115.223999,A 93.1196976,B -40.9738007,C 89.8636017,S 2,T 3}
DECL LDAT LL_OLP20={VEL 2.0,ACC 23.0,APO_DIST 0.0,APO_FAC 0.0,ORI_TYP #VAR,CIRC_TYP #BASE,JERK_FAC 50.0}
DECL FDAT Fl050={TOOL_NO 4,BASE_NO 2,IPO_FRAME #BASE,POINT2[] " "}
DECL PDAT PP_OLP4={VEL 100.0,ACC 50.0,APO_DIST 0.0}
DECL E6POS Xl050={X 1183.39404,Y -1250.13403,Z 302.403015,A 0.0321005285,B 24.9942207,C 90.0242081,S 18,T 11,E1 0.0,E2 0.0,E3 0.0,E4 0.0,E5 0.0,E6 0.0}
DECL FDAT Fl055={TOOL_NO 4,BASE_NO 2,IPO_FRAME #BASE,POINT2[] " ",TQ_STATE FALSE}
DECL E6POS Xl055={X 1194.81201,Y -804.394226,Z 310.400787,A 16.5380306,B 23.6995697,C 97.4459229,S 18,T 11,E1 0.0,E2 0.0,E3 0.0,E4 0.0,E5 0.0,E6 0.0}
DECL LDAT LL_OLP21={VEL 2.0,ACC 23.0,APO_DIST 0.0,APO_FAC 0.0,ORI_TYP #VAR,CIRC_TYP #BASE,JERK_FAC 50.0}
DECL FDAT Fl060={TOOL_NO 4,BASE_NO 2,IPO_FRAME #BASE,POINT2[] " "}
DECL E6POS Xl060={X 1183.14294,Y -837.340271,Z 77.5867462,A 0.0342403911,B 24.9927406,C 90.0283966,S 18,T 11,E1 0.0,E2 0.0,E3 0.0,E4 0.0,E5 0.0,E6 0.0}
DECL LDAT LL_OLP22={VEL 2.0,ACC 23.0,APO_DIST 0.0,APO_FAC 0.0,ORI_TYP #VAR,CIRC_TYP #BASE,JERK_FAC 50.0}
DECL FDAT FSWP_60_0329={TOOL_NO 4,BASE_NO 2,IPO_FRAME #BASE,POINT2[] " "}
DECL E6POS XSWP_60_0329={X 1200.43396,Y -853.982727,Z 69.7639999,A 0.0341486707,B 24.9937897,C 90.0277786,S 18,T 11,E1 0.0,E2 0.0,E3 0.0,E4 0.0,E5 0.0,E6 0.0}
DECL LDAT LL_OLP23={VEL 2.0,ACC 23.0,APO_DIST 0.0,APO_FAC 0.0,ORI_TYP #VAR,CIRC_TYP #BASE,JERK_FAC 50.0}
DECL FDAT Fl065={TOOL_NO 4,BASE_NO 2,IPO_FRAME #BASE,POINT2[] " "}
DECL E6POS Xl065={X 1281.06006,Y -850.894592,Z 69.1942902,A 0.114633001,B 26.8466702,C 89.6470566,S 18,T 11,E1 0.0,E2 0.0,E3 0.0,E4 0.0,E5 0.0,E6 0.0}
DECL LDAT LL_OLP24={VEL 2.0,ACC 23.0,APO_DIST 0.0,APO_FAC 0.0,ORI_TYP #VAR,CIRC_TYP #BASE,JERK_FAC 50.0}
DECL FDAT Fl070={TOOL_NO 4,BASE_NO 2,IPO_FRAME #BASE,POINT2[] " "}
DECL E6POS Xl070={X 1406.45605,Y -849.653503,Z 66.9644928,A 0.107878901,B 29.8631496,C 89.6457672,S 18,T 11,E1 0.0,E2 0.0,E3 0.0,E4 0.0,E5 0.0,E6 0.0}
DECL LDAT LL_OLP25={VEL 2.0,ACC 23.0,APO_DIST 0.0,APO_FAC 0.0,ORI_TYP #VAR,CIRC_TYP #BASE,JERK_FAC 50.0}
DECL FDAT FSWP_60_0343={TOOL_NO 4,BASE_NO 2,IPO_FRAME #BASE,POINT2[] " "}
DECL E6POS XSWP_60_0343={X 1487.79004,Y -857.041626,Z 69.3559265,A 0.0353154801,B 31.7807503,C 90.0282135,S 18,T 11,E1 0.0,E2 0.0,E3 0.0,E4 0.0,E5 0.0,E6 0.0}
DECL LDAT LL_OLP26={VEL 2.0,ACC 23.0,APO_DIST 0.0,APO_FAC 0.0,ORI_TYP #VAR,CIRC_TYP #BASE,JERK_FAC 50.0}
DECL FDAT FSWP_60_0345={TOOL_NO 4,BASE_NO 2,IPO_FRAME #BASE,POINT2[] " "}
DECL E6POS XSWP_60_0345={X 1509.89294,Y -858.199097,Z 68.8594818,A 0.0356448889,B 31.7804108,C 90.025177,S 18,T 11,E1 0.0,E2 0.0,E3 0.0,E4 0.0,E5 0.0,E6 0.0}
DECL LDAT LL_OLP27={VEL 2.0,ACC 23.0,APO_DIST 0.0,APO_FAC 0.0,ORI_TYP #VAR,CIRC_TYP #BASE,JERK_FAC 50.0}
DECL FDAT Fl075={TOOL_NO 4,BASE_NO 2,IPO_FRAME #BASE,POINT2[] " "}
DECL E6POS Xl075={X 1493.10498,Y -814.673889,Z 73.0533295,A 0.0344165489,B 31.9551201,C 90.0252609,S 18,T 11,E1 0.0,E2 0.0,E3 0.0,E4 0.0,E5 0.0,E6 0.0}
DECL LDAT LL_OLP28={VEL 2.0,ACC 23.0,APO_DIST 0.0,APO_FAC 0.0,ORI_TYP #VAR,CIRC_TYP #BASE,JERK_FAC 50.0}
DECL FDAT Fl080={TOOL_NO 4,BASE_NO 2,IPO_FRAME #BASE,POINT2[] " "}
DECL E6POS Xl080={X 1374.17102,Y -827.280273,Z 405.254608,A 5.33724499,B 26.3535309,C 87.9923172,S 18,T 11,E1 0.0,E2 0.0,E3 0.0,E4 0.0,E5 0.0,E6 0.0}
DECL LDAT LL_OLP29={VEL 2.0,ACC 23.0,APO_DIST 0.0,APO_FAC 0.0,ORI_TYP #VAR,CIRC_TYP #BASE,JERK_FAC 50.0}
DECL FDAT Fl085={TOOL_NO 4,BASE_NO 2,IPO_FRAME #BASE,POINT2[] " "}
DECL E6POS Xl085={X 1500.08899,Y -837.090393,Z 632.51709,A 0.199419707,B -0.0117151504,C 90.9192963,S 18,T 3,E1 0.0,E2 0.0,E3 0.0,E4 0.0,E5 0.0,E6 0.0}
DECL LDAT LL_OLP30={VEL 2.0,ACC 23.0,APO_DIST 0.0,APO_FAC 0.0,ORI_TYP #VAR,CIRC_TYP #BASE,JERK_FAC 50.0}
DECL FDAT FSWP_60_0391={TOOL_NO 4,BASE_NO 2,IPO_FRAME #BASE,POINT2[] " "}
DECL E6POS XSWP_60_0391={X 1523.38403,Y -858.364929,Z 642.120422,A 0.0985539034,B -0.00759117305,C 90.4189377,S 18,T 3,E1 0.0,E2 0.0,E3 0.0,E4 0.0,E5 0.0,E6 0.0}
DECL LDAT LL_OLP31={VEL 2.0,ACC 23.0,APO_DIST 0.0,APO_FAC 0.0,ORI_TYP #VAR,CIRC_TYP #BASE,JERK_FAC 50.0}
DECL FDAT Fl090={TOOL_NO 4,BASE_NO 2,IPO_FRAME #BASE,POINT2[] " "}
DECL E6POS Xl090={X 1499.49695,Y -847.102295,Z 632.604492,A 0.02352334,B 5.99430323,C 90.0244064,S 18,T 11,E1 0.0,E2 0.0,E3 0.0,E4 0.0,E5 0.0,E6 0.0}
DECL LDAT LL_OLP32={VEL 2.0,ACC 23.0,APO_DIST 0.0,APO_FAC 0.0,ORI_TYP #VAR,CIRC_TYP #BASE,JERK_FAC 50.0}
DECL FDAT Fl095={TOOL_NO 4,BASE_NO 2,IPO_FRAME #BASE,POINT2[] " "}
DECL E6POS Xl095={X 1462.25598,Y -846.941711,Z 630.032471,A 0.216927305,B 8.61441422,C 90.0247803,S 18,T 11,E1 0.0,E2 0.0,E3 0.0,E4 0.0,E5 0.0,E6 0.0}
DECL LDAT LL_OLP33={VEL 2.0,ACC 23.0,APO_DIST 0.0,APO_FAC 0.0,ORI_TYP #VAR,CIRC_TYP #BASE,JERK_FAC 50.0}
DECL FDAT Fl100={TOOL_NO 4,BASE_NO 2,IPO_FRAME #BASE,POINT2[] " "}
DECL E6POS Xl100={X 1473.21399,Y -845.553589,Z 700.596924,A 0.0294393394,B 16.9969006,C 90.0254974,S 18,T 11,E1 0.0,E2 0.0,E3 0.0,E4 0.0,E5 0.0,E6 0.0}
DECL LDAT LL_OLP34={VEL 2.0,ACC 23.0,APO_DIST 0.0,APO_FAC 0.0,ORI_TYP #VAR,CIRC_TYP #BASE,JERK_FAC 50.0}
DECL FDAT FSWP_60_0397={TOOL_NO 4,BASE_NO 2,IPO_FRAME #BASE,POINT2[] " "}
DECL E6POS XSWP_60_0397={X 1475.43201,Y -857.77533,Z 707.841492,A 0.0292913094,B 16.9969997,C 90.0257187,S 18,T 11,E1 0.0,E2 0.0,E3 0.0,E4 0.0,E5 0.0,E6 0.0}
DECL LDAT LL_OLP35={VEL 2.0,ACC 23.0,APO_DIST 0.0,APO_FAC 0.0,ORI_TYP #VAR,CIRC_TYP #BASE,JERK_FAC 50.0}
DECL FDAT Fl105={TOOL_NO 4,BASE_NO 2,IPO_FRAME #BASE,POINT2[] " "}
DECL E6POS Xl105={X 1473.85596,Y -850.762817,Z 718.293518,A 0.0290593002,B 16.9969196,C 90.0258102,S 18,T 11,E1 0.0,E2 0.0,E3 0.0,E4 0.0,E5 0.0,E6 0.0}
DECL LDAT LL_OLP36={VEL 2.0,ACC 23.0,APO_DIST 0.0,APO_FAC 0.0,ORI_TYP #VAR,CIRC_TYP #BASE,JERK_FAC 50.0}
DECL FDAT Fl110={TOOL_NO 4,BASE_NO 2,IPO_FRAME #BASE,POINT2[] " "}
DECL E6POS Xl110={X 1466.974,Y -839.170593,Z 758.91333,A 0.0293730106,B 16.9969597,C 90.0265732,S 18,T 11,E1 0.0,E2 0.0,E3 0.0,E4 0.0,E5 0.0,E6 0.0}
DECL LDAT LL_OLP37={VEL 2.0,ACC 23.0,APO_DIST 0.0,APO_FAC 0.0,ORI_TYP #VAR,CIRC_TYP #BASE,JERK_FAC 50.0}
DECL FDAT Fl115={TOOL_NO 4,BASE_NO 2,IPO_FRAME #BASE,POINT2[] " "}
DECL E6POS Xl115={X 1521.64502,Y -850.736389,Z 752.462219,A 0.0279998295,B 16.9968109,C 90.0246887,S 18,T 11,E1 0.0,E2 0.0,E3 0.0,E4 0.0,E5 0.0,E6 0.0}
DECL LDAT LL_OLP38={VEL 2.0,ACC 23.0,APO_DIST 0.0,APO_FAC 0.0,ORI_TYP #VAR,CIRC_TYP #BASE,JERK_FAC 50.0}
DECL FDAT FSWP_60_0401={TOOL_NO 4,BASE_NO 2,IPO_FRAME #BASE,POINT2[] " "}
DECL E6POS XSWP_60_0401={X 1530.81396,Y -856.90033,Z 743.679077,A 0.0253196396,B 16.9986095,C 90.0267792,S 18,T 11,E1 0.0,E2 0.0,E3 0.0,E4 0.0,E5 0.0,E6 0.0}
DECL LDAT LL_OLP39={VEL 2.0,ACC 23.0,APO_DIST 0.0,APO_FAC 0.0,ORI_TYP #VAR,CIRC_TYP #BASE,JERK_FAC 50.0}
DECL FDAT Fl120={TOOL_NO 4,BASE_NO 2,IPO_FRAME #BASE,POINT2[] " "}
DECL E6POS Xl120={X 1512.70703,Y -843.356812,Z 757.494385,A 0.0186595395,B 16.9900303,C 90.0240631,S 18,T 11,E1 0.0,E2 0.0,E3 0.0,E4 0.0,E5 0.0,E6 0.0}
DECL LDAT LL_OLP40={VEL 2.0,ACC 23.0,APO_DIST 0.0,APO_FAC 0.0,ORI_TYP #VAR,CIRC_TYP #BASE,JERK_FAC 50.0}
DECL FDAT Fl125={TOOL_NO 4,BASE_NO 2,IPO_FRAME #BASE,POINT2[] " "}
DECL E6POS Xl125={X 1434.79504,Y -838.771729,Z 742.32019,A 0.0195202399,B 19.9976902,C 90.030838,S 18,T 11,E1 0.0,E2 0.0,E3 0.0,E4 0.0,E5 0.0,E6 0.0}
DECL LDAT LL_OLP41={VEL 2.0,ACC 23.0,APO_DIST 0.0,APO_FAC 0.0,ORI_TYP #VAR,CIRC_TYP #BASE,JERK_FAC 50.0}
DECL FDAT Fl130={TOOL_NO 4,BASE_NO 2,IPO_FRAME #BASE,POINT2[] " "}
DECL PDAT PP_OLP5={VEL 100.0,ACC 50.0,APO_DIST 0.0}
DECL E6POS Xl130={X 1277.73901,Y -819.363281,Z 368.684601,A 15.0024996,B 20.6895504,C 95.0901566,S 18,T 11,E1 0.0,E2 0.0,E3 0.0,E4 0.0,E5 0.0,E6 0.0}
DECL FDAT Fl135={TOOL_NO 4,BASE_NO 2,IPO_FRAME #BASE,POINT2[] " "}
DECL PDAT PP_OLP6={VEL 100.0,ACC 100.0,APO_DIST 10.0,APO_MODE #CDIS}
DECL E6POS Xl135={X 1179.62695,Y -846.445313,Z 343.60611,A 16.3660297,B 19.2061691,C 95.5226898,S 18,T 11,E1 0.0,E2 0.0,E3 0.0,E4 0.0,E5 0.0,E6 0.0}
DECL FDAT Fl140={TOOL_NO 4,BASE_NO 2,IPO_FRAME #BASE,POINT2[] " "}
DECL PDAT PP_OLP7={VEL 100.0,ACC 50.0,APO_DIST 0.0}
DECL E6POS Xl140={X 585.392029,Y -2777.80811,Z 1079.05505,A 94.473587,B -14.49792,C 133.0811,S 18,T 11,E1 0.0,E2 0.0,E3 0.0,E4 0.0,E5 0.0,E6 0.0}
DECL FDAT Fl145={TOOL_NO 4,BASE_NO 2,IPO_FRAME #BASE,POINT2[] " "}
DECL PDAT PP_OLP8={VEL 100.0,ACC 100.0,APO_DIST 30.0,APO_MODE #CDIS}
DECL E6POS Xl145={X 1363.80396,Y -1692.80005,Z 601.542725,A 49.0009193,B -3.07281709,C 115.721703,S 18,T 11,E1 0.0,E2 0.0,E3 0.0,E4 0.0,E5 0.0,E6 0.0}
DECL FDAT FLO1679={TOOL_NO 4,BASE_NO 2,IPO_FRAME #BASE,POINT2[] " "}
DECL PDAT PP_OLP9={VEL 100.0,ACC 50.0,APO_DIST 0.0}
DECL BASIS_SUGG_T LAST_BASIS={POINT1[] "P0                      ",POINT2[] "P0                      ",CP_PARAMS[] "CPDAT0                  ",PTP_PARAMS[] "PDAT0                   ",CONT[] "                        ",CP_VEL[] "2.0                     ",PTP_VEL[] " 100                    ",SYNC_PARAMS[] "SYNCDAT                 ",SPL_NAME[] "S0                      "}
DECL PDAT PPDAT1={VEL 100.0,ACC 100.0,APO_DIST 10.0,APO_MODE #CDIS,GEAR_JERK 50.0}
DECL SPOT_SUGG_T LAST_SPOT={GUN[] "1                       ",RETR_CMD[] "#OPN                    ",CHOISE[] "#FIRST                  ",CLO_TM[] "0                       ",PGNO1[] "1                       ",PRESS1[] "0                       ",PGNO2[] "1                       ",PRESS2[] "0                       ",SPOT_PARAMS[] "NORMAL                  "}
DECL PDAT PPDAT12={VEL 100.0,ACC 100.0,APO_DIST 100.0,GEAR_JERK 50.0}
DECL PDAT PPDAT2={VEL 100.0,ACC 100.0,APO_DIST 100.0,GEAR_JERK 50.0}
DECL PDAT PPDAT3={VEL 100.0,ACC 100.0,APO_DIST 100.0,APO_MODE #CDIS,GEAR_JERK 50.0}
DECL PDAT PPDAT4={VEL 100.0,ACC 100.0,APO_DIST 100.0,GEAR_JERK 50.0}
DECL PDAT PPDAT5={VEL 100.0,ACC 100.0,APO_DIST 100.0,GEAR_JERK 50.0}
DECL PDAT PPDAT6={VEL 100.0,ACC 100.0,APO_DIST 100.0,GEAR_JERK 50.0}
DECL E6POS XP1={X 1549.58203,Y -852.089172,Z 995.942017,A 91.1283035,B -67.7504425,C 91.544487,S 18,T 3,E1 0.0,E2 0.0,E3 0.0,E4 0.0,E5 0.0,E6 0.0}
DECL FDAT FP1={TOOL_NO 4,BASE_NO 2,IPO_FRAME #BASE,POINT2[] " ",TQ_STATE FALSE}
DECL PDAT PPDAT7={VEL 100.0,ACC 100.0,APO_DIST 100.0,APO_MODE #CDIS,GEAR_JERK 50.0}
DECL PDAT PPDAT8={VEL 100.0,ACC 100.0,APO_DIST 100.0,GEAR_JERK 50.0}
DECL PDAT PPDAT9={VEL 100.0,ACC 100.0,APO_DIST 100.0,GEAR_JERK 50.0}
DECL PDAT PPDAT10={VEL 100.0,ACC 100.0,APO_DIST 100.0,GEAR_JERK 50.0}
DECL PDAT PPDAT11={VEL 100.0,ACC 100.0,APO_DIST 100.0,APO_MODE #CDIS,GEAR_JERK 50.0}
DECL PDAT PPDAT13={VEL 100.0,ACC 100.0,APO_DIST 100.0,GEAR_JERK 50.0}
DECL E6POS XP2={X 1535.93298,Y -892.826416,Z 444.998413,A 92.6875381,B -41.6146202,C 90.3800812,S 18,T 3,E1 0.0,E2 0.0,E3 0.0,E4 0.0,E5 0.0,E6 0.0}
DECL FDAT FP2={TOOL_NO 4,BASE_NO 2,IPO_FRAME #BASE,POINT2[] " ",TQ_STATE FALSE}
DECL PDAT PPDAT14={VEL 100.0,ACC 80.0,APO_DIST 10.0,APO_MODE #CDIS,GEAR_JERK 50.0}
DECL E6POS XP3={X 1541.92798,Y -889.629089,Z 528.59082,A 92.8173676,B -47.1638908,C 90.296463,S 18,T 3,E1 0.0,E2 0.0,E3 0.0,E4 0.0,E5 0.0,E6 0.0}
DECL FDAT FP3={TOOL_NO 4,BASE_NO 2,IPO_FRAME #BASE,POINT2[] " ",TQ_STATE FALSE}
DECL PDAT PPDAT15={VEL 100.0,ACC 100.0,APO_DIST 100.0,APO_MODE #CDIS,GEAR_JERK 50.0}
DECL PDAT PPDAT16={VEL 100.0,ACC 100.0,APO_DIST 100.0,GEAR_JERK 50.0}
DECL PDAT PPDAT17={VEL 100.0,ACC 100.0,APO_DIST 100.0,GEAR_JERK 50.0}
DECL PDAT PPDAT18={VEL 100.0,ACC 100.0,APO_DIST 100.0,GEAR_JERK 50.0}
DECL PDAT PPDAT19={VEL 100.0,ACC 100.0,APO_DIST 100.0,GEAR_JERK 50.0}
DECL PDAT PPDAT20={VEL 100.0,ACC 100.0,APO_DIST 100.0,GEAR_JERK 50.0}
DECL PDAT PPDAT21={VEL 100.0,ACC 100.0,APO_DIST 10.0,APO_MODE #CDIS,GEAR_JERK 50.0}
DECL PDAT PPDAT22={VEL 100.0,ACC 100.0,APO_DIST 30.0,APO_MODE #CDIS,GEAR_JERK 50.0}
DECL PDAT PPDAT23={VEL 100.0,ACC 100.0,APO_DIST 50.0,APO_MODE #CDIS,GEAR_JERK 50.0}
DECL PDAT PPDAT24={VEL 100.0,ACC 50.0,APO_DIST 0.0,APO_MODE #CDIS,GEAR_JERK 50.0}
DECL PDAT PPDAT25={VEL 100.0,ACC 100.0,APO_DIST 100.0,GEAR_JERK 50.0}
DECL PDAT PPDAT26={VEL 100.0,ACC 100.0,APO_DIST 50.0,APO_MODE #CDIS,GEAR_JERK 50.0}
DECL PDAT PPDAT27={VEL 100.0,ACC 100.0,APO_DIST 50.0,APO_MODE #CDIS,GEAR_JERK 50.0}
DECL PDAT PPDAT28={VEL 100.0,ACC 100.0,APO_DIST 100.0,GEAR_JERK 50.0}
DECL PDAT PPDAT29={VEL 100.0,ACC 100.0,APO_DIST 100.0,GEAR_JERK 50.0}
DECL PDAT PPDAT30={VEL 100.0,ACC 100.0,APO_DIST 50.0,APO_MODE #CDIS,GEAR_JERK 50.0}
DECL PDAT PPDAT31={VEL 100.0,ACC 100.0,APO_DIST 50.0,APO_MODE #CDIS,GEAR_JERK 50.0}
DECL PDAT PPDAT32={VEL 100.0,ACC 100.0,APO_DIST 50.0,APO_MODE #CDIS,GEAR_JERK 50.0}
DECL PDAT PPDAT33={VEL 100.0,ACC 100.0,APO_DIST 100.0,GEAR_JERK 50.0}
DECL PDAT PPDAT34={VEL 100.0,ACC 100.0,APO_DIST 50.0,APO_MODE #CDIS,GEAR_JERK 50.0}
DECL PDAT PPDAT35={VEL 100.0,ACC 100.0,APO_DIST 50.0,APO_MODE #CDIS,GEAR_JERK 50.0}
DECL PDAT PPDAT36={VEL 100.0,ACC 100.0,APO_DIST 100.0,GEAR_JERK 50.0}
DECL PDAT PPDAT37={VEL 100.0,ACC 100.0,APO_DIST 50.0,APO_MODE #CDIS,GEAR_JERK 50.0}
DECL PDAT PPDAT38={VEL 100.0,ACC 100.0,APO_DIST 50.0,APO_MODE #CDIS,GEAR_JERK 50.0}
DECL PDAT PPDAT39={VEL 100.0,ACC 100.0,APO_DIST 50.0,APO_MODE #CDIS,GEAR_JERK 50.0}
DECL PDAT PPDAT40={VEL 100.0,ACC 100.0,APO_DIST 50.0,APO_MODE #CDIS,GEAR_JERK 50.0}
DECL PDAT PPDAT41={VEL 100.0,ACC 100.0,APO_DIST 100.0,GEAR_JERK 50.0}
DECL PDAT PPDAT42={VEL 100.0,ACC 100.0,APO_DIST 10.0,APO_MODE #CDIS,GEAR_JERK 50.0}
DECL PDAT PPDAT43={VEL 100.0,ACC 100.0,APO_DIST 30.0,APO_MODE #CDIS,GEAR_JERK 50.0}
DECL E6POS XP4={X 1021.39502,Y -1375.91895,Z 351.452301,A 0.033490181,B 19.9916191,C 90.0237579,S 18,T 11,E1 0.0,E2 0.0,E3 0.0,E4 0.0,E5 0.0,E6 0.0}
DECL FDAT FP4={TOOL_NO 4,BASE_NO 2,IPO_FRAME #BASE,POINT2[] " ",TQ_STATE FALSE}
DECL PDAT PPDAT44={VEL 100.0,ACC 50.0,APO_DIST 0.0,APO_MODE #CDIS,GEAR_JERK 50.0}
DECL E6POS XP5={X 1257.43103,Y -1225.401,Z 283.898193,A 15.7917099,B 18.8930893,C 95.2303696,S 18,T 11,E1 0.0,E2 0.0,E3 0.0,E4 0.0,E5 0.0,E6 0.0}
DECL FDAT FP5={TOOL_NO 4,BASE_NO 2,IPO_FRAME #BASE,POINT2[] " ",TQ_STATE FALSE}
DECL PDAT PPDAT45={VEL 100.0,ACC 100.0,APO_DIST 30.0,APO_MODE #CDIS,GEAR_JERK 50.0}
DECL E6POS XP6={X 1281.99304,Y -2746.698,Z 868.448303,A 147.915604,B -63.5340195,C 88.4754562,S 18,T 11,E1 0.0,E2 0.0,E3 0.0,E4 0.0,E5 0.0,E6 0.0}
DECL FDAT FP6={TOOL_NO 4,BASE_NO 2,IPO_FRAME #BASE,POINT2[] " ",TQ_STATE FALSE}
DECL PDAT PPDAT46={VEL 100.0,ACC 100.0,APO_DIST 30.0,APO_MODE #CDIS,GEAR_JERK 50.0}
DECL E6POS XP7={X 1233.73901,Y -1125.28296,Z 527.499878,A 37.6324692,B 0.997626424,C 116.177399,S 18,T 11,E1 0.0,E2 0.0,E3 0.0,E4 0.0,E5 0.0,E6 0.0}
DECL FDAT FP7={TOOL_NO 4,BASE_NO 2,IPO_FRAME #BASE,POINT2[] " ",TQ_STATE FALSE}
DECL PDAT PPDAT47={VEL 100.0,ACC 100.0,APO_DIST 50.0,APO_MODE #CDIS,GEAR_JERK 50.0}
DECL E6POS XP8={X 1026.224,Y -2681.75708,Z 608.869812,A 79.3514862,B 3.74117494,C 114.652702,S 18,T 11,E1 0.0,E2 0.0,E3 0.0,E4 0.0,E5 0.0,E6 0.0}
DECL FDAT FP8={TOOL_NO 4,BASE_NO 2,IPO_FRAME #BASE,POINT2[] " ",TQ_STATE FALSE}
DECL PDAT PPDAT48={VEL 100.0,ACC 100.0,APO_DIST 0.0,APO_MODE #CDIS,GEAR_JERK 50.0}
DECL PDAT PPDAT0={VEL 100.0,ACC 100.0,APO_DIST 100.0,GEAR_JERK 50.0}
DECL E6POS XSWP_60_0362={X 1544.04797,Y -894.937378,Z 437.406708,A 92.7001419,B -40.9681511,C 90.4352493,S 18,T 3,E1 0.0,E2 0.0,E3 0.0,E4 0.0,E5 0.0,E6 0.0}
DECL FDAT FSWP_60_0362={TOOL_NO 4,BASE_NO 2,IPO_FRAME #BASE,POINT2[] " "}
DECL LDAT LCPDAT23={VEL 2.0,ACC 100.0,APO_DIST 100.0,APO_FAC 50.0,AXIS_VEL 100.0,AXIS_ACC 100.0,ORI_TYP #VAR,CIRC_TYP #BASE,JERK_FAC 50.0,GEAR_JERK 50.0,EXAX_IGN 0}
DECL E6POS XP9={X 1538.802,Y -894.904175,Z 437.513,A 92.7003632,B -40.9684906,C 90.4346466,S 18,T 3,E1 0.0,E2 0.0,E3 0.0,E4 0.0,E5 0.0,E6 0.0}
DECL FDAT FP9={TOOL_NO 4,BASE_NO 2,IPO_FRAME #BASE,POINT2[] " ",TQ_STATE FALSE}
DECL PDAT PPDAT49={VEL 100.0,ACC 100.0,APO_DIST 100.0,APO_MODE #CDIS,GEAR_JERK 50.0}
DECL E6POS XP10={X 1543.87195,Y -874.356628,Z 769.89563,A 93.3126297,B -63.6034813,C 89.7042007,S 18,T 3,E1 0.0,E2 0.0,E3 0.0,E4 0.0,E5 0.0,E6 0.0}
DECL FDAT FP10={TOOL_NO 4,BASE_NO 2,IPO_FRAME #BASE,POINT2[] " ",TQ_STATE FALSE}
DECL PDAT PPDAT50={VEL 100.0,ACC 100.0,APO_DIST 100.0,APO_MODE #CDIS,GEAR_JERK 50.0}
ENDDAT
